(* IEC 61131-3 sources: AXOpen/src/components.ur.robotics/ctrl/src/AxoUrCb3/v_3_x_x/TypeStructuresAndEnums, 20 files *)

(* ---- eAxoUrRoboticsRobotMode.st ---- *)
NAMESPACE AXOpen.Components.Ur.Robotics
TYPE
    eAxoUrRoboticsRobotMode : USINT
    (

        DISCONNECTED        := USINT#0,
        SAFETY              := USINT#1,
        BOOTING             := USINT#2,
        POWER_OFF           := USINT#3,
       	POWER_ON            := USINT#4,
        IDLE                := USINT#5,
        BACKDRIVE           := USINT#6,
        RUNNING             := USINT#7,
        UPDATING_FIRMWARE   := USINT#8
    );
END_TYPE
END_NAMESPACE

(* ---- AxoUrRobotics_Component_Status.st ---- *)
NAMESPACE AXOpen.Components.Ur.Robotics.v_3_x_x
    {S7.extern=ReadWrite}
    {#ix-attr:[Container(Layout.Stack)]}
    CLASS PUBLIC AxoUrRobotics_Component_Status EXTENDS AXOpen.Components.Robotics.AxoRobot_Status
        VAR PUBLIC
        END_VAR
    END_CLASS
END_NAMESPACE

(* ---- AxoUrRobotics_Config.st ---- *)
NAMESPACE AXOpen.Components.Ur.Robotics.v_3_x_x
    {#ix-attr:[Container(Layout.Stack)]}
    {S7.extern=ReadWrite}
    CLASS PUBLIC AxoUrRobotics_Config
        VAR PUBLIC
            {#ix-set:AttributeName = "<#Info time#>"}
            InfoTime : LTIME := LT#2S;
            {#ix-set:AttributeName = "<#Error time#>"}
            ErrorTime : LTIME := LT#0S;
            {#ix-set:AttributeName = "<#Task timeout#>"}
            TaskTimeout : LTIME := LT#60S;
            {#ix-set:AttributeName = "<#Hardware IDs#>"}
            HWIDs : AxoUrRobotics_HWIDs;
            {#ix-set:AttributeName = "<#Remote power on enabled#>"}
            RemotePowerOnEnabled:BOOL :=FALSE;
            {#ix-set:AttributeName = "<#Remote power on pulse time#>"}
            RemotePowerOnPulse : TIME := T#500MS;
            {#ix-set:AttributeName = "<#IP address#>"}
            IpAddress : STRING;
        END_VAR
    END_CLASS
END_NAMESPACE

(* ---- AxoUrRobotics_Control.st ---- *)
NAMESPACE AXOpen.Components.Ur.Robotics.v_3_x_x
    {S7.extern=ReadWrite}
    {#ix-attr:[Container(Layout.Wrap)]}
    CLASS AxoUrRobotics_Control
        VAR PUBLIC
            {#ix-attr:[Container(Layout.Stack)]}
            {#ix-attr:[Group(GroupLayout.GroupBox)]}
            {#ix-set:AttributeName = "<#Start program#>"}
            Start : BOOL;
            {#ix-set:AttributeName = "<#Stop program#>"}
            Stop : BOOL;
            {#ix-set:AttributeName = "<#Pause program#>"}
            Pause : BOOL;
            {#ix-set:AttributeName = "<#Set motor on#>"}
            MotorOn : BOOL;
            {#ix-set:AttributeName = "<#Run action#>"}
            RunAction : BOOL;

            {#ix-attr:[Container(Layout.Stack)]}
            {#ix-attr:[Group(GroupLayout.GroupBox)]}
            {#ix-set:AttributeName = "<#Master mode#>"}
            MasterMode : BYTE;

            {#ix-attr:[Container(Layout.Stack)]}
            {#ix-attr:[Group(GroupLayout.GroupBox)]}
            {#ix-set:AttributeName = "<#Tool 1 retract#>"}
            Tool_1_Retract : BOOL;
            {#ix-set:AttributeName = "<#Tool 1 extend#>"}
            Tool_1_Extend : BOOL;
            {#ix-set:AttributeName = "<#Tool 2 retract#>"}
            Tool_2_Retract : BOOL;
            {#ix-set:AttributeName = "<#Tool 2 extend#>"}
            Tool_2_Extend : BOOL;
            {#ix-set:AttributeName = "<#Tool 3 retract#>"}
            Tool_3_Retract : BOOL;
            {#ix-set:AttributeName = "<#Tool 3 extend#>"}
            Tool_3_Extend : BOOL;
            {#ix-set:AttributeName = "<#Tool 4 retract#>"}
            Tool_4_Retract : BOOL;
            {#ix-set:AttributeName = "<#Tool 4 extend#>"}
            Tool_4_Extend : BOOL;

            {#ix-attr:[Container(Layout.Stack)]}
            {#ix-attr:[Group(GroupLayout.GroupBox)]}
            {#ix-set:AttributeName = "<#Zones#>"}
            Zone : DINT;
            {#ix-set:AttributeName = "<#In position#>"}
            InPosition : DINT;
            {#ix-set:AttributeName = "<#Action number#>"}
            ActionNo : DINT :=  DINT#255;
            {#ix-set:AttributeName = "<#Global robot speed#>"}
            GlobalSpeed : DINT;
            {#ix-set:AttributeName = "<#Tool number#>"}
            ToolNo : DINT;
            {#ix-set:AttributeName = "<#Workobject number#>"}
            WorkobjectNo : DINT;
            {#ix-set:AttributeName = "<#Point number#>"}
            PointNo : DINT;
            {#ix-set:AttributeName = "<#User specific speed 1#>"}
            UserSpecSpeed1 : REAL;
            {#ix-set:AttributeName = "<#User specific speed 2#>"}
            UserSpecSpeed2 : REAL;

            {#ix-attr:[Container(Layout.Stack)]}
            {#ix-attr:[Group(GroupLayout.GroupBox)]}
            {#ix-set:AttributeName = "<#Coordinates#>"}
            Coordinates : AXOpen.Components.Abstractions.Robotics.AxoRoboticsCoordinates;

            {#ix-attr:[Container(Layout.Wrap)]}
            {#ix-attr:[Group(GroupLayout.GroupBox)]}
            {#ix-set:AttributeName = "<#UR Specific#>"}
            Outputs : AxoUrRoboticsOutputData;
        END_VAR
    END_CLASS
END_NAMESPACE

(* ---- AxoUrRobotics_HWIDs.st ---- *)
NAMESPACE AXOpen.Components.Ur.Robotics.v_3_x_x
    {#ix-attr:[Container(Layout.Stack)]}
    {S7.extern=ReadWrite}
    CLASS PUBLIC AxoUrRobotics_HWIDs
        VAR PUBLIC

            {#ix-set:AttributeName = "<#Hardware ID of the Device#>"}
            HwId_Device                                              : UINT;
            {#ix-set:AttributeName = "<#Hardware ID 'T2O_State' submodule#>"}
            HwId_AxoUrRobotics_T2O_State                             : UINT;
            {#ix-set:AttributeName = "<#Hardware ID 'T2O_IO' submodule#>"}
            HwId_AxoUrRobotics_T2O_IO                                : UINT;
            {#ix-set:AttributeName = "<#Hardware ID 'T2O_Joints' submodule#>"}
            HwId_AxoUrRobotics_T2O_Joints                            : UINT;
            {#ix-set:AttributeName = "<#Hardware ID 'T2O_TCP' submodule#>"}
            HwId_AxoUrRobotics_T2O_TCP                               : UINT;
            {#ix-set:AttributeName = "<#Hardware ID 'T2O_General_Purpose_Bit_Registers' submodule#>"}
            HwId_AxoUrRobotics_T2O_General_Purpose_Bit_Registers     : UINT;
            {#ix-set:AttributeName = "<#Hardware ID 'T2O_General_Purpose_Int_Registers' submodule#>"}
            HwId_AxoUrRobotics_T2O_General_Purpose_Int_Registers     : UINT;
            {#ix-set:AttributeName = "<#Hardware ID 'T2O_General_Purpose_Float_Registers' submodule#>"}
            HwId_AxoUrRobotics_T2O_General_Purpose_Float_Registers   : UINT;
            {#ix-set:AttributeName = "<#Hardware ID 'O2T_Robot_IO' submodule#>"}
            HwId_AxoUrRobotics_O2T_Robot_IO                          : UINT;
            {#ix-set:AttributeName = "<#Hardware ID 'O2T_General_Purpose_Registers_1' submodule#>"}
            HwId_AxoUrRobotics_O2T_General_Purpose_Registers_1       : UINT;
            {#ix-set:AttributeName = "<#Hardware ID 'O2T_General_Purpose_Registers_2' submodule#>"}
            HwId_AxoUrRobotics_O2T_General_Purpose_Registers_2       : UINT;
        END_VAR
    END_CLASS
END_NAMESPACE

(* ---- AxoUrRobotics_O2TIo.st ---- *)
NAMESPACE AXOpen.Components.Ur.Robotics.v_3_x_x
    {#ix-attr:[Container(Layout.Stack)]}
    {S7.extern=ReadWrite}
    CLASS PUBLIC AxoUrRobotics_O2TIo
        VAR PUBLIC
            {#ix-set:AttributeName = "<#Standard digital output mask#>"}
            StandardDigitalOutputMask : USINT;
            {#ix-set:AttributeName = "<#Configurable digital output mask#>"}
            ConfigurableDigitalOutputMask : USINT;
            {#ix-set:AttributeName = "<#Standard digital outputs#>"}
            StandardDigitalOutputs : USINT;
            {#ix-set:AttributeName = "<#Configurable digital outputs#>"}
            ConfigurableDdigitalOutputs : USINT;
            {#ix-set:AttributeName = "<#AOM: Analog output mask#>"}
            AOM_AnalogOutputMask : USINT;
            {#ix-set:AttributeName = "<#AOT: Analog output types#>"}
            AOT_AnalogOutputTypes : USINT;
            {#ix-set:AttributeName = "<#TDOM: Tool digital output mask#>"}
            TDOM_ToolDigitalOutputMask : USINT;
            {#ix-set:AttributeName = "<#TDO: Tool digital output#>"}
            TDO_ToolDigitalOutput : USINT;
            {#ix-set:AttributeName = "<#Standard analog output 0#>"}
            StandardAnalogOutput_0 : REAL;
            {#ix-set:AttributeName = "<#Standard analog output 0#>"}
            StandardAnalogOutput_1 : REAL;
        END_VAR
    END_CLASS
END_NAMESPACE

(* ---- AxoUrRobotics_O2TReg.st ---- *)
NAMESPACE AXOpen.Components.Ur.Robotics.v_3_x_x
    {#ix-attr:[Container(Layout.Stack)]}
    {S7.extern=ReadWrite}
    CLASS PUBLIC AxoUrRobotics_O2TReg
        VAR PUBLIC
            {#ix-set:AttributeName = "<#Bit register 0#>"}
            Bit_0 : BOOL;
            {#ix-set:AttributeName = "<#Bit register 1#>"}
            Bit_1 : BOOL;
            {#ix-set:AttributeName = "<#Bit register 2#>"}
            Bit_2 : BOOL;
            {#ix-set:AttributeName = "<#Bit register 3#>"}
            Bit_3 : BOOL;
            {#ix-set:AttributeName = "<#Bit register 4#>"}
            Bit_4 : BOOL;
            {#ix-set:AttributeName = "<#Bit register 5#>"}
            Bit_5 : BOOL;
            {#ix-set:AttributeName = "<#Bit register 6#>"}
            Bit_6 : BOOL;
            {#ix-set:AttributeName = "<#Bit register 7#>"}
            Bit_7 : BOOL;
            {#ix-set:AttributeName = "<#Bit register 8#>"}
            Bit_8 : BOOL;
            {#ix-set:AttributeName = "<#Bit register 9#>"}
            Bit_9 : BOOL;
            {#ix-set:AttributeName = "<#Bit register 10#>"}
            Bit_10 : BOOL;
            {#ix-set:AttributeName = "<#Bit register 11#>"}
            Bit_11 : BOOL;
            {#ix-set:AttributeName = "<#Bit register 12#>"}
            Bit_12 : BOOL;
            {#ix-set:AttributeName = "<#Bit register 13#>"}
            Bit_13 : BOOL;
            {#ix-set:AttributeName = "<#Bit register 14#>"}
            Bit_14 : BOOL;
            {#ix-set:AttributeName = "<#Bit register 15#>"}
            Bit_15 : BOOL;
            {#ix-set:AttributeName = "<#Bit register 16#>"}
            Bit_16 : BOOL;
            {#ix-set:AttributeName = "<#Bit register 17#>"}
            Bit_17 : BOOL;
            {#ix-set:AttributeName = "<#Bit register 18#>"}
            Bit_18 : BOOL;
            {#ix-set:AttributeName = "<#Bit register 19#>"}
            Bit_19 : BOOL;
            {#ix-set:AttributeName = "<#Bit register 20#>"}
            Bit_20 : BOOL;
            {#ix-set:AttributeName = "<#Bit register 21#>"}
            Bit_21 : BOOL;
            {#ix-set:AttributeName = "<#Bit register 22#>"}
            Bit_22 : BOOL;
            {#ix-set:AttributeName = "<#Bit register 23#>"}
            Bit_23 : BOOL;
            {#ix-set:AttributeName = "<#Bit register 24#>"}
            Bit_24 : BOOL;
            {#ix-set:AttributeName = "<#Bit register 25#>"}
            Bit_25 : BOOL;
            {#ix-set:AttributeName = "<#Bit register 26#>"}
            Bit_26 : BOOL;
            {#ix-set:AttributeName = "<#Bit register 27#>"}
            Bit_27 : BOOL;
            {#ix-set:AttributeName = "<#Bit register 28#>"}
            Bit_28 : BOOL;
            {#ix-set:AttributeName = "<#Bit register 29#>"}
            Bit_29 : BOOL;
            {#ix-set:AttributeName = "<#Bit register 30#>"}
            Bit_30 : BOOL;
            {#ix-set:AttributeName = "<#Bit register 31#>"}
            Bit_31 : BOOL;
            {#ix-set:AttributeName = "<#Int register 0#>"}
            Int_0 : DINT;
            {#ix-set:AttributeName = "<#Int register 1#>"}
            Int_1 : DINT;
            {#ix-set:AttributeName = "<#Int register 2#>"}
            Int_2 : DINT;
            {#ix-set:AttributeName = "<#Int register 3#>"}
            Int_3 : DINT;
            {#ix-set:AttributeName = "<#Int register 4#>"}
            Int_4 : DINT;
            {#ix-set:AttributeName = "<#Int register 5#>"}
            Int_5 : DINT;
            {#ix-set:AttributeName = "<#Int register 6#>"}
            Int_6 : DINT;
            {#ix-set:AttributeName = "<#Int register 7#>"}
            Int_7 : DINT;
            {#ix-set:AttributeName = "<#Int register 8#>"}
            Int_8 : DINT;
            {#ix-set:AttributeName = "<#Int register 9#>"}
            Int_9 : DINT;
            {#ix-set:AttributeName = "<#Int register 10#>"}
            Int_10 : DINT;
            {#ix-set:AttributeName = "<#Int register 11#>"}
            Int_11 : DINT;
            {#ix-set:AttributeName = "<#Float register 0#>"}
            Float_0 : REAL;
            {#ix-set:AttributeName = "<#Float register 1#>"}
            Float_1 : REAL;
            {#ix-set:AttributeName = "<#Float register 2#>"}
            Float_2 : REAL;
            {#ix-set:AttributeName = "<#Float register 3#>"}
            Float_3 : REAL;
            {#ix-set:AttributeName = "<#Float register 4#>"}
            Float_4 : REAL;
            {#ix-set:AttributeName = "<#Float register 5#>"}
            Float_5 : REAL;
            {#ix-set:AttributeName = "<#Float register 6#>"}
            Float_6 : REAL;
            {#ix-set:AttributeName = "<#Float register 7#>"}
            Float_7 : REAL;
            {#ix-set:AttributeName = "<#Float register 8#>"}
            Float_8 : REAL;
            {#ix-set:AttributeName = "<#Float register 9#>"}
            Float_9 : REAL;
            {#ix-set:AttributeName = "<#Float register 10#>"}
            Float_10 : REAL;
            {#ix-set:AttributeName = "<#Float register 11#>"}
            Float_11 : REAL;
        END_VAR
    END_CLASS
END_NAMESPACE

(* ---- AxoUrRobotics_O2TRobot.st ---- *)
NAMESPACE AXOpen.Components.Ur.Robotics.v_3_x_x
    {#ix-attr:[Container(Layout.Stack)]}
    {S7.extern=ReadWrite}
    CLASS PUBLIC AxoUrRobotics_O2TRobot
        VAR PUBLIC
            {#ix-set:AttributeName = "<#SSM: Speed slider fraction mask#>"}
            SSM_SpeedSliderFractionMask : BOOL;
            {#ix-set:AttributeName = "<#Speed slider fraction#>"}
            SpeedSliderFraction : REAL;
        END_VAR
    END_CLASS
END_NAMESPACE

(* ---- AxoUrRobotics_State.st ---- *)
NAMESPACE AXOpen.Components.Ur.Robotics.v_3_x_x
    {S7.extern=ReadWrite}
    {#ix-attr:[Container(Layout.Wrap)]}
    CLASS AxoUrRobotics_State
        VAR PUBLIC
            {#ix-attr:[Container(Layout.Stack)]}
            {#ix-attr:[Group(GroupLayout.GroupBox)]}
            {#ix-set:AttributeName = "<#Robot Mode#>"}
            RobotMode : eAxoUrRoboticsRobotMode;

            {#ix-attr:[Container(Layout.Stack)]}
            {#ix-attr:[Group(GroupLayout.GroupBox)]}
            {#ix-set:AttributeName = "<#In area 1#>"}
            InArea_1 : BOOL;
            {#ix-set:AttributeName = "<#In area 2#>"}
            InArea_2 : BOOL;
            {#ix-set:AttributeName = "<#In area 3#>"}
            InArea_3 : BOOL;
            {#ix-set:AttributeName = "<#In area 4#>"}
            InArea_4 : BOOL;
            {#ix-set:AttributeName = "<#In position 1#>"}
            InPosition_1 : BOOL;
            {#ix-set:AttributeName = "<#In position 2#>"}
            InPosition_2 : BOOL;
            {#ix-set:AttributeName = "<#In position 3#>"}
            InPosition_3 : BOOL;
            {#ix-set:AttributeName = "<#In position 4#>"}
            InPosition_4 : BOOL;

            {#ix-attr:[Container(Layout.Stack)]}
            {#ix-attr:[Group(GroupLayout.GroupBox)]}
            {#ix-set:AttributeName = "<#Zones#>"}
            Zone : DINT;
            {#ix-set:AttributeName = "<#In position#>"}
            InPosition : DINT;

            {#ix-attr:[Container(Layout.Stack)]}
            {#ix-attr:[Group(GroupLayout.GroupBox)]}
            {#ix-set:AttributeName = "<#Tool 1 retract#>"}
            Tool_1_Retract : BOOL;
            {#ix-set:AttributeName = "<#Tool 1 extend#>"}
            Tool_1_Extend : BOOL;
            {#ix-set:AttributeName = "<#Tool 2 retract#>"}
            Tool_2_Retract : BOOL;
            {#ix-set:AttributeName = "<#Tool 2 extend#>"}
            Tool_2_Extend : BOOL;
            {#ix-set:AttributeName = "<#Tool 3 retract#>"}
            Tool_3_Retract : BOOL;
            {#ix-set:AttributeName = "<#Tool 3 extend#>"}
            Tool_3_Extend : BOOL;
            {#ix-set:AttributeName = "<#Tool 4 retract#>"}
            Tool_4_Retract : BOOL;
            {#ix-set:AttributeName = "<#Tool 4 extend#>"}
            Tool_4_Extend : BOOL;

            {#ix-attr:[Container(Layout.Stack)]}
            {#ix-attr:[Group(GroupLayout.GroupBox)]}
            {#ix-set:AttributeName = "<#Action number#>"}
            ActionNo : DINT;
            {#ix-set:AttributeName = "<#Global speed#>"}
            GlobalSpeed : DINT;
            {#ix-set:AttributeName = "<#Tool number#>"}
            ToolNo : DINT;
            {#ix-set:AttributeName = "<#Workobject number#>"}
            WorkobjectNo : DINT;
            {#ix-set:AttributeName = "<#PointNumber#>"}
            PointNo : DINT;
            {#ix-set:AttributeName = "<#User specific speed 1#>"}
            UserSpecSpeed1 : REAL;
            {#ix-set:AttributeName = "<#User specific speed 2#>"}
            UserSpecSpeed2 : REAL;

            {#ix-attr:[Container(Layout.Stack)]}
            {#ix-attr:[Group(GroupLayout.GroupBox)]}
            {#ix-set:AttributeName = "<#Coordinates#>"}
            Coordinates : AXOpen.Components.Abstractions.Robotics.AxoRoboticsCoordinates;

            {#ix-attr:[Container(Layout.Wrap)]}
            {#ix-attr:[Group(GroupLayout.GroupBox)]}
            {#ix-set:AttributeName = "<#UR Specific#>"}
            Inputs:AxoUrRoboticsInputData;
        END_VAR
    END_CLASS
END_NAMESPACE

(* ---- AxoUrRoboticsInputData.st ---- *)
NAMESPACE AXOpen.Components.Ur.Robotics.v_3_x_x
    {#ix-attr:[Container(Layout.Wrap)]}
    {S7.extern=ReadWrite}
    CLASS PUBLIC AxoUrRoboticsInputData
        VAR PUBLIC
            {#ix-attr:[Container(Layout.Stack)]}
            {#ix-attr:[Group(GroupLayout.GroupBox)]}
            {#ix-set:AttributeName = "<#Robot#>"}
            Robot : AxoUrRoboticsT2ORobot;
            {#ix-attr:[Container(Layout.Stack)]}
            {#ix-attr:[Group(GroupLayout.GroupBox)]}
            {#ix-set:AttributeName = "<#State#>"}
            Safety : AxoUrRoboticsT2OSafety;
            {#ix-attr:[Container(Layout.Stack)]}
            {#ix-attr:[Group(GroupLayout.GroupBox)]}
            {#ix-set:AttributeName = "<#IO state#>"}
            IO : AxoUrRoboticsT2OIo;
            {#ix-attr:[Container(Layout.Stack)]}
            {#ix-attr:[Group(GroupLayout.GroupBox)]}
            {#ix-set:AttributeName = "<#Tool state#>"}
            Tool : AxoUrRoboticsT2OTool;
            {#ix-attr:[Container(Layout.Stack)]}
            {#ix-attr:[Group(GroupLayout.GroupBox)]}
            {#ix-set:AttributeName = "<#Joints#>"}
            Joints : AxoUrRoboticsT2OJoints;
            {#ix-attr:[Container(Layout.Stack)]}
            {#ix-attr:[Group(GroupLayout.GroupBox)]}
            {#ix-set:AttributeName = "<#TCP#>"}
            TCP : AxoUrRoboticsT2OTcp;
            {#ix-attr:[Container(Layout.Stack)]}
            {#ix-attr:[Group(GroupLayout.GroupBox)]}
            {#ix-set:AttributeName = "<#Bits#>"}
            Bits : AxoUrRoboticsT2OBitRegs;
            {#ix-attr:[Container(Layout.Stack)]}
            {#ix-attr:[Group(GroupLayout.GroupBox)]}
            {#ix-set:AttributeName = "<#Ints#>"}
            Ints : AxoUrRoboticsT2OIntRegs;
            {#ix-attr:[Container(Layout.Stack)]}
            {#ix-attr:[Group(GroupLayout.GroupBox)]}
            {#ix-set:AttributeName = "<#Floats#>"}
            Floats : AxoUrRoboticsT2OFloatRegs;
        END_VAR
    END_CLASS
END_NAMESPACE

(* ---- AxoUrRoboticsOutputData.st ---- *)
NAMESPACE AXOpen.Components.Ur.Robotics.v_3_x_x
    {#ix-attr:[Container(Layout.Wrap)]}
    {S7.extern=ReadWrite}
    CLASS PUBLIC AxoUrRoboticsOutputData
        VAR PUBLIC
            {#ix-attr:[Container(Layout.Stack)]}
            {#ix-attr:[Group(GroupLayout.GroupBox)]}
            {#ix-set:AttributeName = "<#Speed#>"}
            Speed   :   AxoUrRobotics_O2TRobot;
            {#ix-attr:[Container(Layout.Stack)]}
            {#ix-attr:[Group(GroupLayout.GroupBox)]}
            {#ix-set:AttributeName = "<#IO#>"}
            IO      :   AxoUrRobotics_O2TIo;
            {#ix-attr:[Container(Layout.Stack)]}
            {#ix-attr:[Group(GroupLayout.GroupBox)]}
            {#ix-set:AttributeName = "<#Reg 1#>"}
            Reg1    :   AxoUrRobotics_O2TReg;
            {#ix-attr:[Container(Layout.Stack)]}
            {#ix-attr:[Group(GroupLayout.GroupBox)]}
            {#ix-set:AttributeName = "<#Reg 2#>"}
            Reg2    :   AxoUrRobotics_O2TReg;
        END_VAR
    END_CLASS
END_NAMESPACE

(* ---- AxoUrRoboticsT2OBitRegs.st ---- *)
NAMESPACE AXOpen.Components.Ur.Robotics.v_3_x_x
    {#ix-attr:[Container(Layout.Stack)]}
    {S7.extern=ReadWrite}
    CLASS PUBLIC AxoUrRoboticsT2OBitRegs
        VAR PUBLIC
            {#ix-set:AttributeName = "<#Bit register 0#>"}
            Register_0 : BOOL;
            {#ix-set:AttributeName = "<#Bit register 1#>"}
            Register_1 : BOOL;
            {#ix-set:AttributeName = "<#Bit register 2#>"}
            Register_2 : BOOL;
            {#ix-set:AttributeName = "<#Bit register 3#>"}
            Register_3 : BOOL;
            {#ix-set:AttributeName = "<#Bit register 4#>"}
            Register_4 : BOOL;
            {#ix-set:AttributeName = "<#Bit register 5#>"}
            Register_5 : BOOL;
            {#ix-set:AttributeName = "<#Bit register 6#>"}
            Register_6 : BOOL;
            {#ix-set:AttributeName = "<#Bit register 7#>"}
            Register_7 : BOOL;
            {#ix-set:AttributeName = "<#Bit register 8#>"}
            Register_8 : BOOL;
            {#ix-set:AttributeName = "<#Bit register 9#>"}
            Register_9 : BOOL;
            {#ix-set:AttributeName = "<#Bit register 10#>"}
            Register_10 : BOOL;
            {#ix-set:AttributeName = "<#Bit register 11#>"}
            Register_11 : BOOL;
            {#ix-set:AttributeName = "<#Bit register 12#>"}
            Register_12 : BOOL;
            {#ix-set:AttributeName = "<#Bit register 13#>"}
            Register_13 : BOOL;
            {#ix-set:AttributeName = "<#Bit register 14#>"}
            Register_14 : BOOL;
            {#ix-set:AttributeName = "<#Bit register 15#>"}
            Register_15 : BOOL;
            {#ix-set:AttributeName = "<#Bit register 16#>"}
            Register_16 : BOOL;
            {#ix-set:AttributeName = "<#Bit register 17#>"}
            Register_17 : BOOL;
            {#ix-set:AttributeName = "<#Bit register 18#>"}
            Register_18 : BOOL;
            {#ix-set:AttributeName = "<#Bit register 19#>"}
            Register_19 : BOOL;
            {#ix-set:AttributeName = "<#Bit register 20#>"}
            Register_20 : BOOL;
            {#ix-set:AttributeName = "<#Bit register 21#>"}
            Register_21 : BOOL;
            {#ix-set:AttributeName = "<#Bit register 22#>"}
            Register_22 : BOOL;
            {#ix-set:AttributeName = "<#Bit register 23#>"}
            Register_23 : BOOL;
            {#ix-set:AttributeName = "<#Bit register 24#>"}
            Register_24 : BOOL;
            {#ix-set:AttributeName = "<#Bit register 25#>"}
            Register_25 : BOOL;
            {#ix-set:AttributeName = "<#Bit register 26#>"}
            Register_26 : BOOL;
            {#ix-set:AttributeName = "<#Bit register 27#>"}
            Register_27 : BOOL;
            {#ix-set:AttributeName = "<#Bit register 28#>"}
            Register_28 : BOOL;
            {#ix-set:AttributeName = "<#Bit register 29#>"}
            Register_29 : BOOL;
            {#ix-set:AttributeName = "<#Bit register 30#>"}
            Register_30 : BOOL;
            {#ix-set:AttributeName = "<#Bit register 31#>"}
            Register_31 : BOOL;
            {#ix-set:AttributeName = "<#Bit register 32#>"}
            Register_32 : BOOL;
            {#ix-set:AttributeName = "<#Bit register 33#>"}
            Register_33 : BOOL;
            {#ix-set:AttributeName = "<#Bit register 34#>"}
            Register_34 : BOOL;
            {#ix-set:AttributeName = "<#Bit register 35#>"}
            Register_35 : BOOL;
            {#ix-set:AttributeName = "<#Bit register 36#>"}
            Register_36 : BOOL;
            {#ix-set:AttributeName = "<#Bit register 37#>"}
            Register_37 : BOOL;
            {#ix-set:AttributeName = "<#Bit register 38#>"}
            Register_38 : BOOL;
            {#ix-set:AttributeName = "<#Bit register 39#>"}
            Register_39 : BOOL;
            {#ix-set:AttributeName = "<#Bit register 40#>"}
            Register_40 : BOOL;
            {#ix-set:AttributeName = "<#Bit register 41#>"}
            Register_41 : BOOL;
            {#ix-set:AttributeName = "<#Bit register 42#>"}
            Register_42 : BOOL;
            {#ix-set:AttributeName = "<#Bit register 43#>"}
            Register_43 : BOOL;
            {#ix-set:AttributeName = "<#Bit register 44#>"}
            Register_44 : BOOL;
            {#ix-set:AttributeName = "<#Bit register 45#>"}
            Register_45 : BOOL;
            {#ix-set:AttributeName = "<#Bit register 46#>"}
            Register_46 : BOOL;
            {#ix-set:AttributeName = "<#Bit register 47#>"}
            Register_47 : BOOL;
            {#ix-set:AttributeName = "<#Bit register 48#>"}
            Register_48 : BOOL;
            {#ix-set:AttributeName = "<#Bit register 49#>"}
            Register_49 : BOOL;
            {#ix-set:AttributeName = "<#Bit register 50#>"}
            Register_50 : BOOL;
            {#ix-set:AttributeName = "<#Bit register 51#>"}
            Register_51 : BOOL;
            {#ix-set:AttributeName = "<#Bit register 52#>"}
            Register_52 : BOOL;
            {#ix-set:AttributeName = "<#Bit register 53#>"}
            Register_53 : BOOL;
            {#ix-set:AttributeName = "<#Bit register 54#>"}
            Register_54 : BOOL;
            {#ix-set:AttributeName = "<#Bit register 55#>"}
            Register_55 : BOOL;
            {#ix-set:AttributeName = "<#Bit register 56#>"}
            Register_56 : BOOL;
            {#ix-set:AttributeName = "<#Bit register 57#>"}
            Register_57 : BOOL;
            {#ix-set:AttributeName = "<#Bit register 58#>"}
            Register_58 : BOOL;
            {#ix-set:AttributeName = "<#Bit register 59#>"}
            Register_59 : BOOL;
            {#ix-set:AttributeName = "<#Bit register 60#>"}
            Register_60 : BOOL;
            {#ix-set:AttributeName = "<#Bit register 61#>"}
            Register_61 : BOOL;
            {#ix-set:AttributeName = "<#Bit register 62#>"}
            Register_62 : BOOL;
            {#ix-set:AttributeName = "<#Bit register 63#>"}
            Register_63 : BOOL;
        END_VAR
    END_CLASS
END_NAMESPACE

(* ---- AxoUrRoboticsT2OFloatRegs.st ---- *)
NAMESPACE AXOpen.Components.Ur.Robotics.v_3_x_x
    {#ix-attr:[Container(Layout.Stack)]}
    {S7.extern=ReadWrite}
    CLASS PUBLIC AxoUrRoboticsT2OFloatRegs
        VAR PUBLIC
            {#ix-set:AttributeName = "<#Float register 0#>"}
            Register_0 : REAL;
            {#ix-set:AttributeName = "<#Float register 1#>"}
            Register_1 : REAL;
            {#ix-set:AttributeName = "<#Float register 2#>"}
            Register_2 : REAL;
            {#ix-set:AttributeName = "<#Float register 3#>"}
            Register_3 : REAL;
            {#ix-set:AttributeName = "<#Float register 4#>"}
            Register_4 : REAL;
            {#ix-set:AttributeName = "<#Float register 5#>"}
            Register_5 : REAL;
            {#ix-set:AttributeName = "<#Float register 6#>"}
            Register_6 : REAL;
            {#ix-set:AttributeName = "<#Float register 7#>"}
            Register_7 : REAL;
            {#ix-set:AttributeName = "<#Float register 8#>"}
            Register_8 : REAL;
            {#ix-set:AttributeName = "<#Float register 9#>"}
            Register_9 : REAL;
            {#ix-set:AttributeName = "<#Float register 10#>"}
            Register_10 : REAL;
            {#ix-set:AttributeName = "<#Float register 11#>"}
            Register_11 : REAL;
            {#ix-set:AttributeName = "<#Float register 12#>"}
            Register_12 : REAL;
            {#ix-set:AttributeName = "<#Float register 13#>"}
            Register_13 : REAL;
            {#ix-set:AttributeName = "<#Float register 14#>"}
            Register_14 : REAL;
            {#ix-set:AttributeName = "<#Float register 15#>"}
            Register_15 : REAL;
            {#ix-set:AttributeName = "<#Float register 16#>"}
            Register_16 : REAL;
            {#ix-set:AttributeName = "<#Float register 17#>"}
            Register_17 : REAL;
            {#ix-set:AttributeName = "<#Float register 18#>"}
            Register_18 : REAL;
            {#ix-set:AttributeName = "<#Float register 19#>"}
            Register_19 : REAL;
            {#ix-set:AttributeName = "<#Float register 20#>"}
            Register_20 : REAL;
            {#ix-set:AttributeName = "<#Float register 21#>"}
            Register_21 : REAL;
            {#ix-set:AttributeName = "<#Float register 22#>"}
            Register_22 : REAL;
            {#ix-set:AttributeName = "<#Float register 23#>"}
            Register_23 : REAL;
        END_VAR
    END_CLASS
END_NAMESPACE

(* ---- AxoUrRoboticsT2OIntRegs.st ---- *)
NAMESPACE AXOpen.Components.Ur.Robotics.v_3_x_x
    {#ix-attr:[Container(Layout.Stack)]}
    {S7.extern=ReadWrite}
    CLASS PUBLIC AxoUrRoboticsT2OIntRegs
        VAR PUBLIC
            {#ix-set:AttributeName = "<#Int register 0#>"}
            Register_0 : DINT;
            {#ix-set:AttributeName = "<#Int register 1#>"}
            Register_1 : DINT;
            {#ix-set:AttributeName = "<#Int register 2#>"}
            Register_2 : DINT;
            {#ix-set:AttributeName = "<#Int register 3#>"}
            Register_3 : DINT;
            {#ix-set:AttributeName = "<#Int register 4#>"}
            Register_4 : DINT;
            {#ix-set:AttributeName = "<#Int register 5#>"}
            Register_5 : DINT;
            {#ix-set:AttributeName = "<#Int register 6#>"}
            Register_6 : DINT;
            {#ix-set:AttributeName = "<#Int register 7#>"}
            Register_7 : DINT;
            {#ix-set:AttributeName = "<#Int register 8#>"}
            Register_8 : DINT;
            {#ix-set:AttributeName = "<#Int register 9#>"}
            Register_9 : DINT;
            {#ix-set:AttributeName = "<#Int register 10#>"}
            Register_10 : DINT;
            {#ix-set:AttributeName = "<#Int register 11#>"}
            Register_11 : DINT;
            {#ix-set:AttributeName = "<#Int register 12#>"}
            Register_12 : DINT;
            {#ix-set:AttributeName = "<#Int register 13#>"}
            Register_13 : DINT;
            {#ix-set:AttributeName = "<#Int register 14#>"}
            Register_14 : DINT;
            {#ix-set:AttributeName = "<#Int register 15#>"}
            Register_15 : DINT;
            {#ix-set:AttributeName = "<#Int register 16#>"}
            Register_16 : DINT;
            {#ix-set:AttributeName = "<#Int register 17#>"}
            Register_17 : DINT;
            {#ix-set:AttributeName = "<#Int register 18#>"}
            Register_18 : DINT;
            {#ix-set:AttributeName = "<#Int register 19#>"}
            Register_19 : DINT;
            {#ix-set:AttributeName = "<#Int register 20#>"}
            Register_20 : DINT;
            {#ix-set:AttributeName = "<#Int register 21#>"}
            Register_21 : DINT;
            {#ix-set:AttributeName = "<#Int register 22#>"}
            Register_22 : DINT;
            {#ix-set:AttributeName = "<#Int register 23#>"}
            Register_23 : DINT;
        END_VAR
    END_CLASS
END_NAMESPACE

(* ---- AxoUrRoboticsT2OIo.st ---- *)
NAMESPACE AXOpen.Components.Ur.Robotics.v_3_x_x
    {#ix-attr:[Container(Layout.Stack)]}
    {S7.extern=ReadWrite}
    CLASS PUBLIC AxoUrRoboticsT2OIo
        VAR PUBLIC
            {#ix-set:AttributeName = "<#Standard digital inputs#>"}
            StandardDigitalInputs : USINT;
            {#ix-set:AttributeName = "<#Configurable digital inputs#>"}
            ConfigurableDigitalInputs : USINT;
            {#ix-set:AttributeName = "<#Standard digital outputs#>"}
            StandardDigitalOutputs : USINT;
            {#ix-set:AttributeName = "<#Configurable digital outputs#>"}
            ConfigurableDigitalOutputs : USINT;
            {#ix-set:AttributeName = "<#Analog I/O types#>"}
            AnalogIoTypes : USINT;
            {#ix-set:AttributeName = "<#Standard analog input 0 [A or V]#>"}
            StandardAnalogInput_0 : REAL;
            {#ix-set:AttributeName = "<#Standard analog input 1 [A or V]#>"}
            StandardAnalogInput_1 : REAL;
            {#ix-set:AttributeName = "<#Standard analog output 0 [A or V]#>"}
            StandardAnalogOutput_0 : REAL;
            {#ix-set:AttributeName = "<#Standard analog output 1 [A or V]#>"}
            StandardAnalogOutput_1 : REAL;
            {#ix-set:AttributeName = "<#I/O current [A]#>"}
            Current : REAL;
            {#ix-set:AttributeName = "<#Euromap67 input bit 0#>"}
            Euromap67InputBit_0 : BOOL;
            {#ix-set:AttributeName = "<#Euromap67 input bit 1#>"}
            Euromap67InputBit_1 : BOOL;
            {#ix-set:AttributeName = "<#Euromap67 input bit 2#>"}
            Euromap67InputBit_2 : BOOL;
            {#ix-set:AttributeName = "<#Euromap67 input bit 3#>"}
            Euromap67InputBit_3 : BOOL;
            {#ix-set:AttributeName = "<#Euromap67 input bit 4#>"}
            Euromap67InputBit_4 : BOOL;
            {#ix-set:AttributeName = "<#Euromap67 input bit 5#>"}
            Euromap67InputBit_5 : BOOL;
            {#ix-set:AttributeName = "<#Euromap67 input bit 6#>"}
            Euromap67InputBit_6 : BOOL;
            {#ix-set:AttributeName = "<#Euromap67 input bit 7#>"}
            Euromap67InputBit_7 : BOOL;
            {#ix-set:AttributeName = "<#Euromap67 input bit 8#>"}
            Euromap67InputBit_8 : BOOL;
            {#ix-set:AttributeName = "<#Euromap67 input bit 9#>"}
            Euromap67InputBit_9 : BOOL;
            {#ix-set:AttributeName = "<#Euromap67 input bit 10#>"}
            Euromap67InputBit_10 : BOOL;
            {#ix-set:AttributeName = "<#Euromap67 input bit 11#>"}
            Euromap67InputBit_11 : BOOL;
            {#ix-set:AttributeName = "<#Euromap67 input bit 12#>"}
            Euromap67InputBit_12 : BOOL;
            {#ix-set:AttributeName = "<#Euromap67 input bit 13#>"}
            Euromap67InputBit_13 : BOOL;
            {#ix-set:AttributeName = "<#Euromap67 input bit 14#>"}
            Euromap67InputBit_14 : BOOL;
            {#ix-set:AttributeName = "<#Euromap67 input bit 15#>"}
            Euromap67InputBit_15 : BOOL;
            {#ix-set:AttributeName = "<#Euromap67 input bit 16#>"}
            Euromap67InputBit_16 : BOOL;
            {#ix-set:AttributeName = "<#Euromap67 input bit 17#>"}
            Euromap67InputBit_17 : BOOL;
            {#ix-set:AttributeName = "<#Euromap67 input bit 18#>"}
            Euromap67InputBit_18 : BOOL;
            {#ix-set:AttributeName = "<#Euromap67 input bit 19#>"}
            Euromap67InputBit_19 : BOOL;
            {#ix-set:AttributeName = "<#Euromap67 input bit 20#>"}
            Euromap67InputBit_20 : BOOL;
            {#ix-set:AttributeName = "<#Euromap67 input bit 21#>"}
            Euromap67InputBit_21 : BOOL;
            {#ix-set:AttributeName = "<#Euromap67 input bit 22#>"}
            Euromap67InputBit_22 : BOOL;
            {#ix-set:AttributeName = "<#Euromap67 input bit 23#>"}
            Euromap67InputBit_23 : BOOL;
            {#ix-set:AttributeName = "<#Euromap67 input bit 24#>"}
            Euromap67InputBit_24 : BOOL;
            {#ix-set:AttributeName = "<#Euromap67 input bit 25#>"}
            Euromap67InputBit_25 : BOOL;
            {#ix-set:AttributeName = "<#Euromap67 input bit 26#>"}
            Euromap67InputBit_26 : BOOL;
            {#ix-set:AttributeName = "<#Euromap67 input bit 27#>"}
            Euromap67InputBit_27 : BOOL;
            {#ix-set:AttributeName = "<#Euromap67 input bit 28#>"}
            Euromap67InputBit_28 : BOOL;
            {#ix-set:AttributeName = "<#Euromap67 input bit 29#>"}
            Euromap67InputBit_29 : BOOL;
            {#ix-set:AttributeName = "<#Euromap67 input bit 30#>"}
            Euromap67InputBit_30 : BOOL;
            {#ix-set:AttributeName = "<#Euromap67 input bit 31#>"}
            Euromap67InputBit_31 : BOOL;
            {#ix-set:AttributeName = "<#Euromap67 input bit 32#>"}
            Euromap67InputBit_32 : BOOL;
            {#ix-set:AttributeName = "<#Euromap67 output bit 0#>"}
            Euromap67outputBit_0 : BOOL;
            {#ix-set:AttributeName = "<#Euromap67 output bit 1#>"}
            Euromap67outputBit_1 : BOOL;
            {#ix-set:AttributeName = "<#Euromap67 output bit 2#>"}
            Euromap67outputBit_2 : BOOL;
            {#ix-set:AttributeName = "<#Euromap67 output bit 3#>"}
            Euromap67outputBit_3 : BOOL;
            {#ix-set:AttributeName = "<#Euromap67 output bit 4#>"}
            Euromap67outputBit_4 : BOOL;
            {#ix-set:AttributeName = "<#Euromap67 output bit 5#>"}
            Euromap67outputBit_5 : BOOL;
            {#ix-set:AttributeName = "<#Euromap67 output bit 6#>"}
            Euromap67outputBit_6 : BOOL;
            {#ix-set:AttributeName = "<#Euromap67 output bit 7#>"}
            Euromap67outputBit_7 : BOOL;
            {#ix-set:AttributeName = "<#Euromap67 output bit 8#>"}
            Euromap67outputBit_8 : BOOL;
            {#ix-set:AttributeName = "<#Euromap67 output bit 9#>"}
            Euromap67outputBit_9 : BOOL;
            {#ix-set:AttributeName = "<#Euromap67 output bit 10#>"}
            Euromap67outputBit_10 : BOOL;
            {#ix-set:AttributeName = "<#Euromap67 output bit 11#>"}
            Euromap67outputBit_11 : BOOL;
            {#ix-set:AttributeName = "<#Euromap67 output bit 12#>"}
            Euromap67outputBit_12 : BOOL;
            {#ix-set:AttributeName = "<#Euromap67 output bit 13#>"}
            Euromap67outputBit_13 : BOOL;
            {#ix-set:AttributeName = "<#Euromap67 output bit 14#>"}
            Euromap67outputBit_14 : BOOL;
            {#ix-set:AttributeName = "<#Euromap67 output bit 15#>"}
            Euromap67outputBit_15 : BOOL;
            {#ix-set:AttributeName = "<#Euromap67 output bit 16#>"}
            Euromap67outputBit_16 : BOOL;
            {#ix-set:AttributeName = "<#Euromap67 output bit 17#>"}
            Euromap67outputBit_17 : BOOL;
            {#ix-set:AttributeName = "<#Euromap67 output bit 18#>"}
            Euromap67outputBit_18 : BOOL;
            {#ix-set:AttributeName = "<#Euromap67 output bit 19#>"}
            Euromap67outputBit_19 : BOOL;
            {#ix-set:AttributeName = "<#Euromap67 output bit 20#>"}
            Euromap67outputBit_20 : BOOL;
            {#ix-set:AttributeName = "<#Euromap67 output bit 21#>"}
            Euromap67outputBit_21 : BOOL;
            {#ix-set:AttributeName = "<#Euromap67 output bit 22#>"}
            Euromap67outputBit_22 : BOOL;
            {#ix-set:AttributeName = "<#Euromap67 output bit 23#>"}
            Euromap67outputBit_23 : BOOL;
            {#ix-set:AttributeName = "<#Euromap67 output bit 24#>"}
            Euromap67outputBit_24 : BOOL;
            {#ix-set:AttributeName = "<#Euromap67 output bit 25#>"}
            Euromap67outputBit_25 : BOOL;
            {#ix-set:AttributeName = "<#Euromap67 output bit 26#>"}
            Euromap67outputBit_26 : BOOL;
            {#ix-set:AttributeName = "<#Euromap67 output bit 27#>"}
            Euromap67outputBit_27 : BOOL;
            {#ix-set:AttributeName = "<#Euromap67 output bit 28#>"}
            Euromap67outputBit_28 : BOOL;
            {#ix-set:AttributeName = "<#Euromap67 output bit 29#>"}
            Euromap67outputBit_29 : BOOL;
            {#ix-set:AttributeName = "<#Euromap67 output bit 30#>"}
            Euromap67outputBit_30 : BOOL;
            {#ix-set:AttributeName = "<#Euromap67 output bit 31#>"}
            Euromap67outputBit_31 : BOOL;
            {#ix-set:AttributeName = "<#Euromap67 output bit 32#>"}
            Euromap67outputBit_32 : BOOL;
            {#ix-set:AttributeName = "<#Euromap67 24V voltage#>"}
            Euromap6724Voltage : REAL;
            {#ix-set:AttributeName = "<#Euromap67 24V current#>"}
            Euromap6724VCurrent : REAL;
        END_VAR
    END_CLASS
END_NAMESPACE

(* ---- AxoUrRoboticsT2OJoints.st ---- *)
NAMESPACE AXOpen.Components.Ur.Robotics.v_3_x_x
    {#ix-attr:[Container(Layout.Stack)]}
    {S7.extern=ReadWrite}
    CLASS PUBLIC AxoUrRoboticsT2OJoints
        VAR PUBLIC
            {#ix-set:AttributeName = "<#Joint position 0 [rad]#>"}
            JointPosition_0 : REAL;
            {#ix-set:AttributeName = "<#Joint position 1 [rad]#>"}
            JointPosition_1 : REAL;
            {#ix-set:AttributeName = "<#Joint position 2 [rad]#>"}
            JointPosition_2 : REAL;
            {#ix-set:AttributeName = "<#Joint position 3 [rad]#>"}
            JointPosition_3 : REAL;
            {#ix-set:AttributeName = "<#Joint position 4 [rad]#>"}
            JointPosition_4 : REAL;
            {#ix-set:AttributeName = "<#Joint position 5 [rad]#>"}
            JointPosition_5 : REAL;
            {#ix-set:AttributeName = "<#Joint velocity 0 [rad/s]#>"}
            JointVelocity_0 : REAL;
            {#ix-set:AttributeName = "<#Joint velocity 1 [rad/s]#>"}
            JointVelocity_1 : REAL;
            {#ix-set:AttributeName = "<#Joint velocity 2 [rad/s]#>"}
            JointVelocity_2 : REAL;
            {#ix-set:AttributeName = "<#Joint velocity 3 [rad/s]#>"}
            JointVelocity_3 : REAL;
            {#ix-set:AttributeName = "<#Joint velocity 4 [rad/s]#>"}
            JointVelocity_4 : REAL;
            {#ix-set:AttributeName = "<#Joint velocity 5 [rad/s]#>"}
            JointVelocity_5 : REAL;
            {#ix-set:AttributeName = "<#Joint current 0 [A]#>"}
            JointCurrent_0 : REAL;
            {#ix-set:AttributeName = "<#Joint current 1 [A]#>"}
            JointCurrent_1 : REAL;
            {#ix-set:AttributeName = "<#Joint current 2 [A]#>"}
            JointCurrent_2 : REAL;
            {#ix-set:AttributeName = "<#Joint current 3 [A]#>"}
            JointCurrent_3 : REAL;
            {#ix-set:AttributeName = "<#Joint current 4 [A]#>"}
            JointCurrent_4 : REAL;
            {#ix-set:AttributeName = "<#Joint current 5 [A]#>"}
            JointCurrent_5 : REAL;
            {#ix-set:AttributeName = "<#Joint temperature 0 [°C]#>"}
            JointTemperature_0 : REAL;
            {#ix-set:AttributeName = "<#Joint temperature 1 [°C]#>"}
            JointTemperature_1 : REAL;
            {#ix-set:AttributeName = "<#Joint temperature 2 [°C]#>"}
            JointTemperature_2 : REAL;
            {#ix-set:AttributeName = "<#Joint temperature 3 [°C]#>"}
            JointTemperature_3 : REAL;
            {#ix-set:AttributeName = "<#Joint temperature 4 [°C]#>"}
            JointTemperature_4 : REAL;
            {#ix-set:AttributeName = "<#Joint temperature 5 [°C]#>"}
            JointTemperature_5 : REAL;
            {#ix-set:AttributeName = "<#Joint mode 0#>"}
            JointMode_0 : USINT;
            {#ix-set:AttributeName = "<#Joint mode 1#>"}
            JointMode_1 : USINT;
            {#ix-set:AttributeName = "<#Joint mode 2#>"}
            JointMode_2 : USINT;
            {#ix-set:AttributeName = "<#Joint mode 3#>"}
            JointMode_3 : USINT;
            {#ix-set:AttributeName = "<#Joint mode 4#>"}
            JointMode_4 : USINT;
            {#ix-set:AttributeName = "<#Joint mode 5#>"}
            JointMode_5 : USINT;
        END_VAR
    END_CLASS
END_NAMESPACE

(* ---- AxoUrRoboticsT2ORobot.st ---- *)
NAMESPACE AXOpen.Components.Ur.Robotics.v_3_x_x
    {#ix-attr:[Container(Layout.Stack)]}
    {S7.extern=ReadWrite}
    CLASS PUBLIC AxoUrRoboticsT2ORobot
        VAR PUBLIC
            {#ix-set:AttributeName = "<#Controller major version#>"}
            ControllerMajorVersion : USINT;
            {#ix-set:AttributeName = "<#Controller minor version#>"}
            ControllerMinorVersion : USINT;
            {#ix-set:AttributeName = "<#Reserved#>"}
            Reserved : UINT;
            {#ix-set:AttributeName = "<#Robot mode#>"}
            RobotMode : USINT;
            {#ix-set:AttributeName = "<#Real time machine seconds#>"}
            RealtimeMachineSeconds : USINT;
            {#ix-set:AttributeName = "<#Real time machine milliseconds#>"}
            RealtimeMachineMilliseconds : UINT;
            {#ix-set:AttributeName = "<#Real time machine minutes#>"}
            RealtimeMachineMinutes : USINT;
            {#ix-set:AttributeName = "<#Real time machine hours#>"}
            RealtimeMachineHours : USINT;
            {#ix-set:AttributeName = "<#Real time machine days#>"}
            RealtimeMachineDays : UINT;
            {#ix-set:AttributeName = "<#Robot current [A]#>"}
            RobotCurrent : REAL;
            {#ix-set:AttributeName = "<#PW: Is power on#>"}
            PW_IsPowerOn : BOOL;
            {#ix-set:AttributeName = "<#PR: Is program running#>"}
            PR_IsProgramRunning : BOOL;
            {#ix-set:AttributeName = "<#TB: Is teach button pressed#>"}
            TB_IsTeachButtonPressed : BOOL;
            {#ix-set:AttributeName = "<#PB: Is power button pressed#>"}
            PB_IsPowerButtonPressed : BOOL;
            {#ix-set:AttributeName = "<#Speed slider fraction#>"}
            SpeedSliderFraction : REAL;
        END_VAR
    END_CLASS
END_NAMESPACE

(* ---- AxoUrRoboticsT2OSafety.st ---- *)
NAMESPACE AXOpen.Components.Ur.Robotics.v_3_x_x
    {#ix-attr:[Container(Layout.Stack)]}
    {S7.extern=ReadWrite}
    CLASS PUBLIC AxoUrRoboticsT2OSafety
        VAR PUBLIC
            {#ix-set:AttributeName = "<#Safety mode#>"}
            SafetyMode : USINT;
            {#ix-set:AttributeName = "<#NO: Is normal mode#>"}
            NO_IsNormalMode : BOOL;
            {#ix-set:AttributeName = "<#RD: Is reduced mode#>"}
            RD_IsReducedMode : BOOL;
            {#ix-set:AttributeName = "<#PS: Is protective stopped#>"}
            PS_IsProtectiveStopped : BOOL;
            {#ix-set:AttributeName = "<#RC: Is recovery mode#>"}
            RC_IsRecoveryMode : BOOL;
            {#ix-set:AttributeName = "<#SS: Is safeguard stopped#>"}
            SS_IsSafeguardStopped : BOOL;
            {#ix-set:AttributeName = "<#SES: Is system emergency stopped#>"}
            SES_IsSystemEmergencyStopped : BOOL;
            {#ix-set:AttributeName = "<#RES: Is robot emergency stopped#>"}
            RES_IsRobotEmergencyStopped : BOOL;
            {#ix-set:AttributeName = "<#ES: Is emergency stopped#>"}
            ES_IsEmergencyStopped : BOOL;
            {#ix-set:AttributeName = "<#VL: Is violation#>"}
            VL_IsViolation : BOOL;
            {#ix-set:AttributeName = "<#FT: Is fault#>"}
            FT_IsFault : BOOL;
            {#ix-set:AttributeName = "<#ST: Is stopped due TO safety#>"}
            ST_IsStoppedDueSafety : BOOL;
        END_VAR
    END_CLASS
END_NAMESPACE

(* ---- AxoUrRoboticsT2OTcp.st ---- *)
NAMESPACE AXOpen.Components.Ur.Robotics.v_3_x_x
    {#ix-attr:[Container(Layout.Stack)]}
    {S7.extern=ReadWrite}
    CLASS PUBLIC AxoUrRoboticsT2OTcp
        VAR PUBLIC
            {#ix-set:AttributeName = "<#Actual TCP Position#>"}
            Postition : AXOpen.Components.Abstractions.Robotics.AxoRoboticsCoordinates;
            {#ix-set:AttributeName = "<#Actual TCP Velocity#>"}
            Velocity : AXOpen.Components.Abstractions.Robotics.AxoRoboticsCoordinates;
            {#ix-set:AttributeName = "<#Actual TCP Force#>"}
            Force : AXOpen.Components.Abstractions.Robotics.AxoRoboticsBasicCoordinates;
            {#ix-set:AttributeName = "<#Actual TCP Torque#>"}
            Torque : AXOpen.Components.Abstractions.Robotics.AxoRoboticsBasicCoordinates;
            {#ix-set:AttributeName = "<#TCP force scalar [N]#>"}
            TCP_ForceScalar : REAL;
        END_VAR
    END_CLASS
END_NAMESPACE

(* ---- AxoUrRoboticsT2OTool.st ---- *)
NAMESPACE AXOpen.Components.Ur.Robotics.v_3_x_x
    {#ix-attr:[Container(Layout.Stack)]}
    {S7.extern=ReadWrite}
    CLASS PUBLIC AxoUrRoboticsT2OTool
        VAR PUBLIC
            {#ix-set:AttributeName = "<#Tool mode#>"}
            ToolMode : USINT;
            {#ix-set:AttributeName = "<#TDI: Tool Digital Inputs#>"}
            TDI_ToolDigitalInputs : USINT;
            {#ix-set:AttributeName = "<#TDO: Tool Digital Outputs#>"}
            TDO_ToolDigitalOutputs : USINT;
            {#ix-set:AttributeName = "<#TAIT: Tool Analog Input Types#>"}
            TAIT_ToolAnalogInputTypes : USINT;
            {#ix-set:AttributeName = "<#Tool analog input 0 [A OR V]#>"}
            ToolAnalogInput_0: REAL;
            {#ix-set:AttributeName = "<#Tool analog input 1 [A OR V]#>"}
            ToolAnalogInput_1: REAL;
            {#ix-set:AttributeName = "<#Tool output voltage [V]#>"}
            ToolOutputVoltage : REAL;
            {#ix-set:AttributeName = "<#Tool current [A]#>"}
            ToolCurrent : REAL;
        END_VAR
    END_CLASS
END_NAMESPACE
